FUNCTION_BLOCK Basis EXTENDS GrundstrukturSkill
VAR_INPUT
END_VAR
VAR_OUTPUT
END_VAR
VAR
END_VAR

IF bFehler THEN
	iState := 3;
END_IF

CASE iState OF 
0: 	// BEREIT
		// DO
		iSkillCommand := 0;
		
		IF bExecute THEN
			iSkillCommand := 1;																							// Starten des Objektes 
		END_IF	
		
		IF iObjState = 3 THEN
			bStarten := TRUE;
		END_IF
			
		// TRANSITION	
		IF bStarten THEN
			bStarten := FALSE;
			iState := 1;																							// Objekt wurde gestartet
		END_IF
// _________________________________________________________________________________________________________________________
1: 	// LAUFEND
		// DO
		iSkillCommand := 0;
		bBusy := TRUE;																									// Skill wird ausgeführt
		
		IF bTargetReached OR bLimitReached THEN																			// Prüfen ob Prozessziel erreicht wurde
			iSkillCommand := 2;
		END_IF
		
		IF iSysCommand := 3 THEN																						// Transition wenn System das Orbjekt stoppt
			bBusy := FALSE;																									// Skill wird nicht mehr ausgeführt
			bStoppen := TRUE;
		END_IF
		
		IF iObjState = 4 THEN																							// Objekt hat Prozess abgeschlossen
			bBusy := FALSE;																									// Skill wird nicht mehr ausgeführt
			bObjektFertig := TRUE;																							// Objekt ist fertig und wieder bereit
		END_IF
		
		IF bLimitReached AND iObjState = 5 THEN																			// Objekt wurde duch Skill gestoppt - LIMIT
			iSkillCommand := 0;																								// Zurücksetzen von Command
			bLimitReached := FALSE;																							// Zurücksetzen von Information	
			bBusy := FALSE;																									// Skill wird nicht mehr ausgeführt
			bLimitErreicht := TRUE;	
		END_IF
		
		IF bTargetReached AND iObjState = 5 THEN																			// Objekt wurde duch Skill gestoppt - LIMIT
			iSkillCommand := 0;																									// Zurücksetzen von Command
			bTargetReached := FALSE;																							// Zurücksetzen von Information	
			bBusy := FALSE;																										// Skill wird nicht mehr ausgeführt
			bWertErreicht := TRUE;	
		END_IF
			
		// TRANSITION 
		IF bStoppen THEN																								// Transition zu BEREIT
			bStoppen := FALSE;																							
			iState := 0;
		END_IF
		
		IF bObjektFertig THEN																							// Transition zu ABGESCHLOSSEN
			bObjektFertig := FALSE;																							// Skill wird nicht mehr ausgeführt
			iState := 2;																									// Objekt ist fertig und wieder bereit
		END_IF
		
		IF bLimitErreicht THEN																							// Transition zu LIMIT
			bLimitErreicht := FALSE;
			iState := 4;
		END_IF
		
		IF bWertErreicht THEN																							// Transition zu ERREICHT																						// Skill wird nicht mehr ausgeführt
			bWertErreicht := FALSE;
			iState := 5;
		END_IF
			
// _________________________________________________________________________________________________________________________			
2: 	// ABGESCHLOSSEN
		// DO
		bDone := TRUE;																									// Skill wurde erfolgreich ausgeführt
			
		iSkillCommand := 3;																								// Objekt resetten
		
		IF iObjState = 1 THEN																							// Objekt wurde geresettet
			iSkillCommand := 0;																								// Zurücksetzen von Command
			bDone := FALSE;																									// Zurücksetzen von Skill
			bSkillFertig := TRUE;									
		END_IF
			
		//  TRANSITION
		IF bSkillFertig THEN
			bSkillFertig := FALSE;																																											// Resetten von Objekt
			iState := 0;
		END_IF
		
// _________________________________________________________________________________________________________________________
3: 	// FEHLER
		// DO 	
		iSkillCommand := 0;
		
		bDone := FALSE;
		bBusy := FALSE;
		
		IF iSysCommand := 4 THEN
			bResetten := TRUE;
		END_IF
		
		// TRANSITION
		IF bResetten THEN
			bResetten := FALSE;
			iState := 0;
		END_IF
		
// _________________________________________________________________________________________________________________________			
4: 	// LIMIT
		// DO 
		iSkillCommand := 0;
		bLimit := TRUE;																									// Limit wurde erreicht
		
		iSkillCommand := 3;																								// Objekt resetten
		
		IF iSysCommand := 4 THEN
			iSkillCommand := 3;																							// Objekt resetten
		END_IF
		
		IF iObjState = 1 THEN																							// Objekt wurde geresettet
			iSkillCommand := 0;																								// Zurücksetzen von Command
			bDone := FALSE;																									// Zurücksetzen von Skill
			bResetten := TRUE;								
		END_IF
	
		// TRANSITION
		IF bResetten THEN
			bResetten := FALSE;
			bLimit := FALSE;																							// Zurücksetzen von Output-Variable
			iSkillCommand := 3;																							// Resetten von Objekt 
			iState := 0;
		END_IF
			
// _________________________________________________________________________________________________________________________
5: 	// ERREICHT		
		// DO 
		iSkillCommand := 0;
		bDone := TRUE;																									// Skill wurde erfolgreich ausgeführt
		
		iSkillCommand := 3;																								// Objekt resetten
		
		IF iObjState = 1 THEN																							// Objekt wurde geresettet
			iSkillCommand := 0;																								// Zurücksetzen von Command
			bDone := FALSE;																									// Zurücksetzen von Skill
			bSkillFertig := TRUE;									
		END_IF
		
		// TRANSITION
		IF bSkillFertig THEN
			bSkillFertig := FALSE;
			bLimit := FALSE;																							// Zurücksetzen von Output-Variable
			iSkillCommand := 3;																							// Resetten von Objekt 
			iState := 0;
		END_IF
		
END_CASE

END_FUNCTION_BLOCK

(* stored: Version 1.1.0.1
   POU Basis: Id {13b7da4f-c74a-4c94-87fb-63c919ff396f}, SpecialFunc None *)
